// TIA Portal V19 export
FUNCTION_BLOCK "F_Zone10_FB"   // FB115, F_LAD
TITLE = SAFETY ZONE 10 - AREA 01 (MATERIAL FEEDING A01)
// stored: Access Published
   VAR
      D07 : "Door_FB";
      FNS : "ForceNormalStop";
      F_Sinamics_Straightener : "FDevice_Sinamics_FB";
      Cumulative_Feed_TwoHands_SafeMotion { ExternalAccessible := 'False'; ExternalVisible := 'False'; ExternalWritable := 'False'} : Bool;
   END_VAR
   VAR_TEMP
      DoorNormalStop : Bool;
      DoorSafeStop : Bool;
      DoorOpened : Bool;
   END_VAR
   VAR CONSTANT
      STRAIGHTENER_S120_STOPPING_TIME : Time := t#3s;
   END_VAR
BEGIN

REGION Network 1: < < < < < < < < < < DOOR > > > > > > > > > >
END_REGION

REGION Network 2: Zone Entry enable
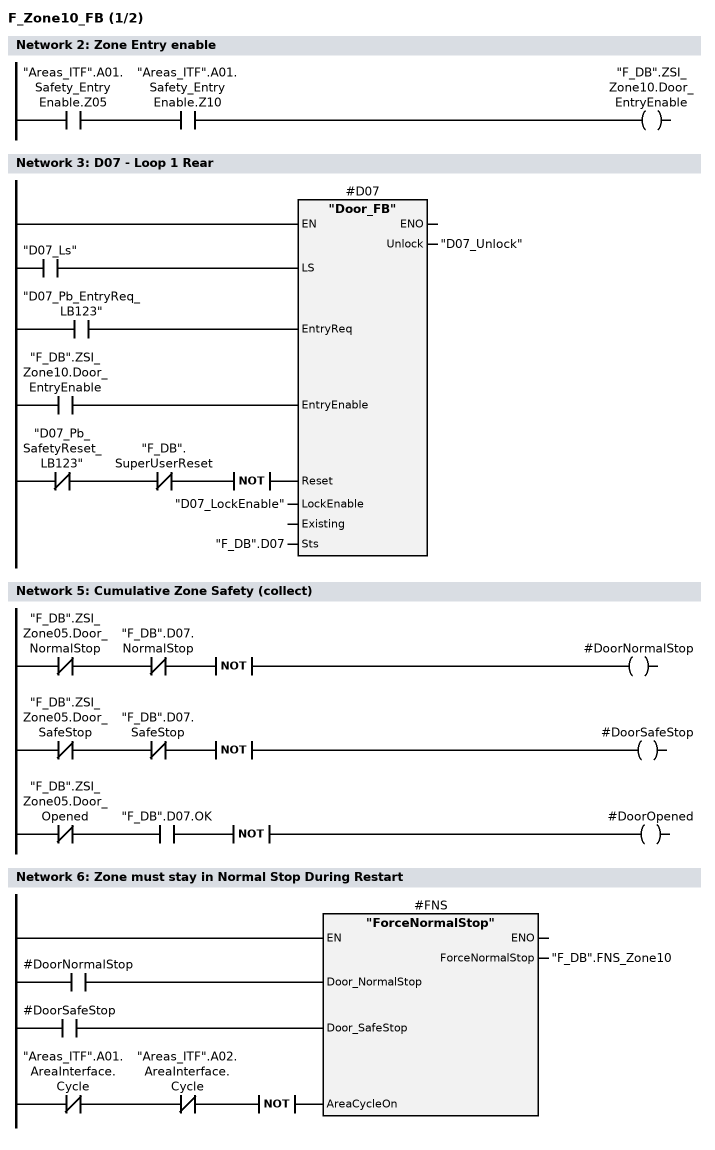
   RUNG wire#powerrail
      Contact( "Areas_ITF".A01.Safety_EntryEnable.Z05 )
      Contact( "Areas_ITF".A01.Safety_EntryEnable.Z10 )
      Coil( "F_DB".ZSI_Zone10.Door_EntryEnable )
   END_RUNG
   // the same network as SCL:
   "F_DB".ZSI_Zone10.Door_EntryEnable := "Areas_ITF".A01.Safety_EntryEnable.Z05 AND "Areas_ITF".A01.Safety_EntryEnable.Z10;
END_REGION

REGION Network 3: D07 - Loop 1 Rear
   RUNG wire#powerrail
      #D07(LS := wire#w1, EntryReq := wire#w2, EntryEnable := wire#w3, Reset := wire#w4, LockEnable := "D07_LockEnable", Existing :=, Sts := "F_DB".D07, Unlock => "D07_Unlock")
   END_RUNG
   RUNG wire#powerrail
      Contact( "D07_Ls" )
   END_RUNG wire#w1
   RUNG wire#powerrail
      Contact( "D07_Pb_EntryReq_LB123" )
   END_RUNG wire#w2
   RUNG wire#powerrail
      Contact( "F_DB".ZSI_Zone10.Door_EntryEnable )
   END_RUNG wire#w3
   RUNG wire#powerrail
      I_Contact( "D07_Pb_SafetyReset_LB123" )
      I_Contact( "F_DB".SuperUserReset )
      Not()
   END_RUNG wire#w4
   // the same network as SCL:
   #D07(LS := "D07_Ls",   // "Door_FB"
        EntryReq := "D07_Pb_EntryReq_LB123",
        EntryEnable := "F_DB".ZSI_Zone10.Door_EntryEnable,
        Reset := NOT (NOT "D07_Pb_SafetyReset_LB123" AND NOT "F_DB".SuperUserReset),
        LockEnable := "D07_LockEnable",
        Sts := "F_DB".D07,
        Unlock => "D07_Unlock");
END_REGION

REGION Network 4: < < < < < < < < < < ZONE SAFETY INTERFACE > > > > > > > > > >
END_REGION

REGION Network 5: Cumulative Zone Safety (collect)
   RUNG wire#powerrail
      I_Contact( "F_DB".ZSI_Zone05.Door_NormalStop )
      I_Contact( "F_DB".D07.NormalStop )
      Not()
      Coil( #DoorNormalStop )
   END_RUNG
   RUNG wire#powerrail
      I_Contact( "F_DB".ZSI_Zone05.Door_SafeStop )
      I_Contact( "F_DB".D07.SafeStop )
      Not()
      Coil( #DoorSafeStop )
   END_RUNG
   RUNG wire#powerrail
      I_Contact( "F_DB".ZSI_Zone05.Door_Opened )
      Contact( "F_DB".D07.OK )
      Not()
      Coil( #DoorOpened )
   END_RUNG
   // the same network as SCL:
   #DoorNormalStop := NOT (NOT "F_DB".ZSI_Zone05.Door_NormalStop AND NOT "F_DB".D07.NormalStop);
   #DoorSafeStop := NOT (NOT "F_DB".ZSI_Zone05.Door_SafeStop AND NOT "F_DB".D07.SafeStop);
   #DoorOpened := NOT (NOT "F_DB".ZSI_Zone05.Door_Opened AND "F_DB".D07.OK);
END_REGION

REGION Network 6: Zone must stay in Normal Stop During Restart
   RUNG wire#powerrail
      #FNS(Door_NormalStop := wire#w1, Door_SafeStop := wire#w2, AreaCycleOn := wire#w3, ForceNormalStop => "F_DB".FNS_Zone10)
   END_RUNG
   RUNG wire#powerrail
      Contact( #DoorNormalStop )
   END_RUNG wire#w1
   RUNG wire#powerrail
      Contact( #DoorSafeStop )
   END_RUNG wire#w2
   RUNG wire#powerrail
      I_Contact( "Areas_ITF".A01.AreaInterface.Cycle )
      I_Contact( "Areas_ITF".A02.AreaInterface.Cycle )
      Not()
   END_RUNG wire#w3
   // the same network as SCL:
   #FNS(Door_NormalStop := #DoorNormalStop,   // "ForceNormalStop"
        Door_SafeStop := #DoorSafeStop,
        AreaCycleOn := NOT (NOT "Areas_ITF".A01.AreaInterface.Cycle AND NOT "Areas_ITF".A02.AreaInterface.Cycle),
        ForceNormalStop => "F_DB".FNS_Zone10);
END_REGION

REGION Network 7: Cumulative Zone Safety
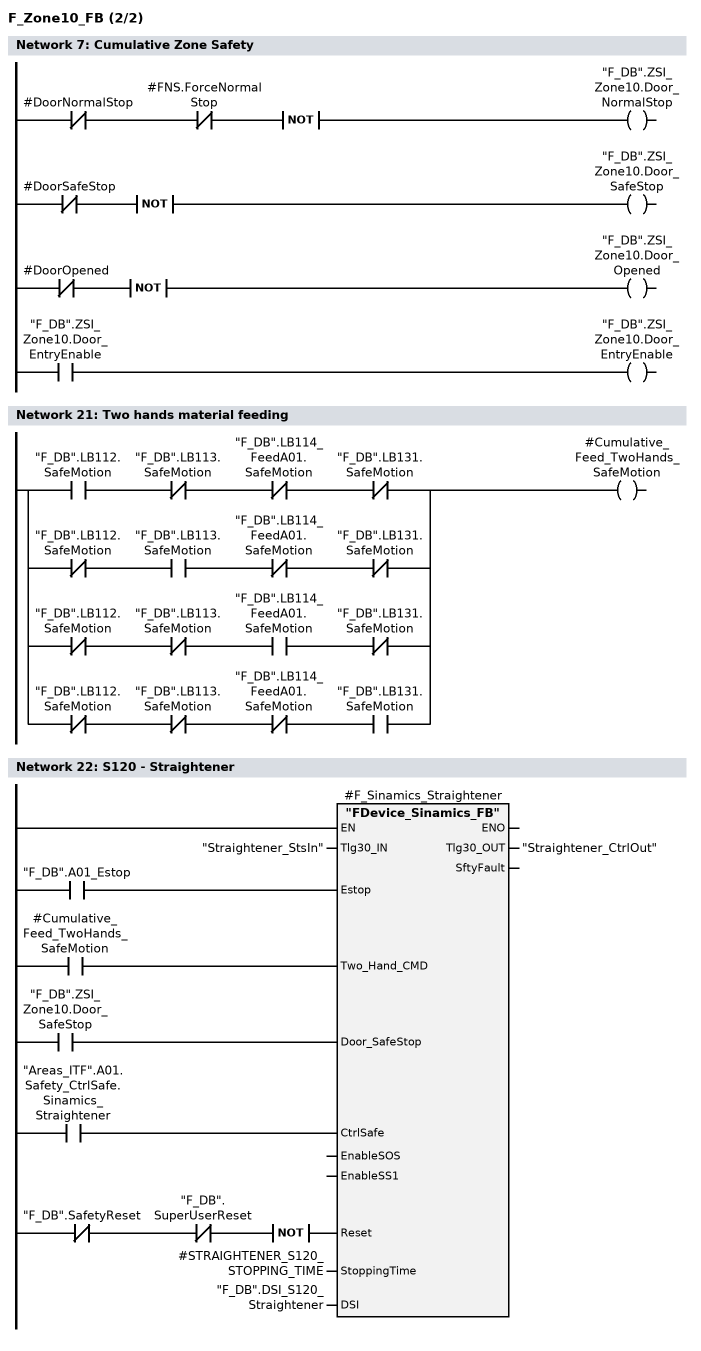
   RUNG wire#powerrail
      I_Contact( #DoorNormalStop )
      I_Contact( #FNS.ForceNormalStop )
      Not()
      Coil( "F_DB".ZSI_Zone10.Door_NormalStop )
   END_RUNG
   RUNG wire#powerrail
      I_Contact( #DoorSafeStop )
      Not()
      Coil( "F_DB".ZSI_Zone10.Door_SafeStop )
   END_RUNG
   RUNG wire#powerrail
      I_Contact( #DoorOpened )
      Not()
      Coil( "F_DB".ZSI_Zone10.Door_Opened )
   END_RUNG
   RUNG wire#powerrail
      Contact( "F_DB".ZSI_Zone10.Door_EntryEnable )
      Coil( "F_DB".ZSI_Zone10.Door_EntryEnable )
   END_RUNG
   // the same network as SCL:
   "F_DB".ZSI_Zone10.Door_NormalStop := NOT (NOT #DoorNormalStop AND NOT #FNS.ForceNormalStop);
   "F_DB".ZSI_Zone10.Door_SafeStop := NOT (NOT #DoorSafeStop);
   "F_DB".ZSI_Zone10.Door_Opened := NOT (NOT #DoorOpened);
   "F_DB".ZSI_Zone10.Door_EntryEnable := "F_DB".ZSI_Zone10.Door_EntryEnable;
END_REGION

REGION Network 8: >
END_REGION

REGION Network 9: >
END_REGION

REGION Network 10: >
END_REGION

REGION Network 11: < < < < < < < < < < DEVICES SAFETY VALVES > > > > > > > > > >
END_REGION

REGION Network 12: >
END_REGION

REGION Network 13: >
END_REGION

REGION Network 14: >
END_REGION

REGION Network 15: < < < < < < < < < < DEVICES CONTACTORS > > > > > > > > > >
END_REGION

REGION Network 16: >
END_REGION

REGION Network 17: >
END_REGION

REGION Network 18: >
END_REGION

REGION Network 19: >
END_REGION

REGION Network 20: < < < < < < < < < < DEVICES S120 > > > > > > > > > >
END_REGION

REGION Network 21: Two hands material feeding
   RUNG wire#powerrail
      Contact( "F_DB".LB112.SafeMotion )
      I_Contact( "F_DB".LB113.SafeMotion )
      I_Contact( "F_DB".LB114_FeedA01.SafeMotion )
      I_Contact( "F_DB".LB131.SafeMotion )
      wire#w1
      Coil( #Cumulative_Feed_TwoHands_SafeMotion )
   END_RUNG
   RUNG wire#powerrail
      I_Contact( "F_DB".LB112.SafeMotion )
      Contact( "F_DB".LB113.SafeMotion )
      I_Contact( "F_DB".LB114_FeedA01.SafeMotion )
      I_Contact( "F_DB".LB131.SafeMotion )
   END_RUNG wire#w1
   RUNG wire#powerrail
      I_Contact( "F_DB".LB112.SafeMotion )
      I_Contact( "F_DB".LB113.SafeMotion )
      Contact( "F_DB".LB114_FeedA01.SafeMotion )
      I_Contact( "F_DB".LB131.SafeMotion )
   END_RUNG wire#w1
   RUNG wire#powerrail
      I_Contact( "F_DB".LB112.SafeMotion )
      I_Contact( "F_DB".LB113.SafeMotion )
      I_Contact( "F_DB".LB114_FeedA01.SafeMotion )
      Contact( "F_DB".LB131.SafeMotion )
   END_RUNG wire#w1
   // the same network as SCL:
   #Cumulative_Feed_TwoHands_SafeMotion := ("F_DB".LB112.SafeMotion AND NOT "F_DB".LB113.SafeMotion AND NOT "F_DB".LB114_FeedA01.SafeMotion AND NOT "F_DB".LB131.SafeMotion) OR (NOT "F_DB".LB112.SafeMotion AND "F_DB".LB113.SafeMotion AND NOT "F_DB".LB114_FeedA01.SafeMotion AND NOT "F_DB".LB131.SafeMotion) OR (NOT "F_DB".LB112.SafeMotion AND NOT "F_DB".LB113.SafeMotion AND "F_DB".LB114_FeedA01.SafeMotion AND NOT "F_DB".LB131.SafeMotion) OR (NOT "F_DB".LB112.SafeMotion AND NOT "F_DB".LB113.SafeMotion AND NOT "F_DB".LB114_FeedA01.SafeMotion AND "F_DB".LB131.SafeMotion);
END_REGION

REGION Network 22: S120 - Straightener
   RUNG wire#powerrail
      #F_Sinamics_Straightener(Estop := wire#w1, Two_Hand_CMD := wire#w2, Door_SafeStop := wire#w3, CtrlSafe := wire#w4, Reset := wire#w5, Tlg30_IN := "Straightener_StsIn", EnableSOS :=, EnableSS1 :=, StoppingTime := #STRAIGHTENER_S120_STOPPING_TIME, DSI := "F_DB".DSI_S120_Straightener, Tlg30_OUT => "Straightener_CtrlOut", SftyFault =>)
   END_RUNG
   RUNG wire#powerrail
      Contact( "F_DB".A01_Estop )
   END_RUNG wire#w1
   RUNG wire#powerrail
      Contact( #Cumulative_Feed_TwoHands_SafeMotion )
   END_RUNG wire#w2
   RUNG wire#powerrail
      Contact( "F_DB".ZSI_Zone10.Door_SafeStop )
   END_RUNG wire#w3
   RUNG wire#powerrail
      Contact( "Areas_ITF".A01.Safety_CtrlSafe.Sinamics_Straightener )
   END_RUNG wire#w4
   RUNG wire#powerrail
      I_Contact( "F_DB".SafetyReset )
      I_Contact( "F_DB".SuperUserReset )
      Not()
   END_RUNG wire#w5
   // the same network as SCL:
   #F_Sinamics_Straightener(Tlg30_IN := "Straightener_StsIn",   // "FDevice_Sinamics_FB"
                           Estop := "F_DB".A01_Estop,
                           Two_Hand_CMD := #Cumulative_Feed_TwoHands_SafeMotion,
                           Door_SafeStop := "F_DB".ZSI_Zone10.Door_SafeStop,
                           CtrlSafe := "Areas_ITF".A01.Safety_CtrlSafe.Sinamics_Straightener,
                           Reset := NOT (NOT "F_DB".SafetyReset AND NOT "F_DB".SuperUserReset),
                           StoppingTime := #STRAIGHTENER_S120_STOPPING_TIME,
                           DSI := "F_DB".DSI_S120_Straightener,
                           Tlg30_OUT => "Straightener_CtrlOut");
END_REGION

REGION Network 23: >
END_REGION

REGION Network 24: >
END_REGION

REGION Network 25: >
END_REGION
END_FUNCTION_BLOCK
